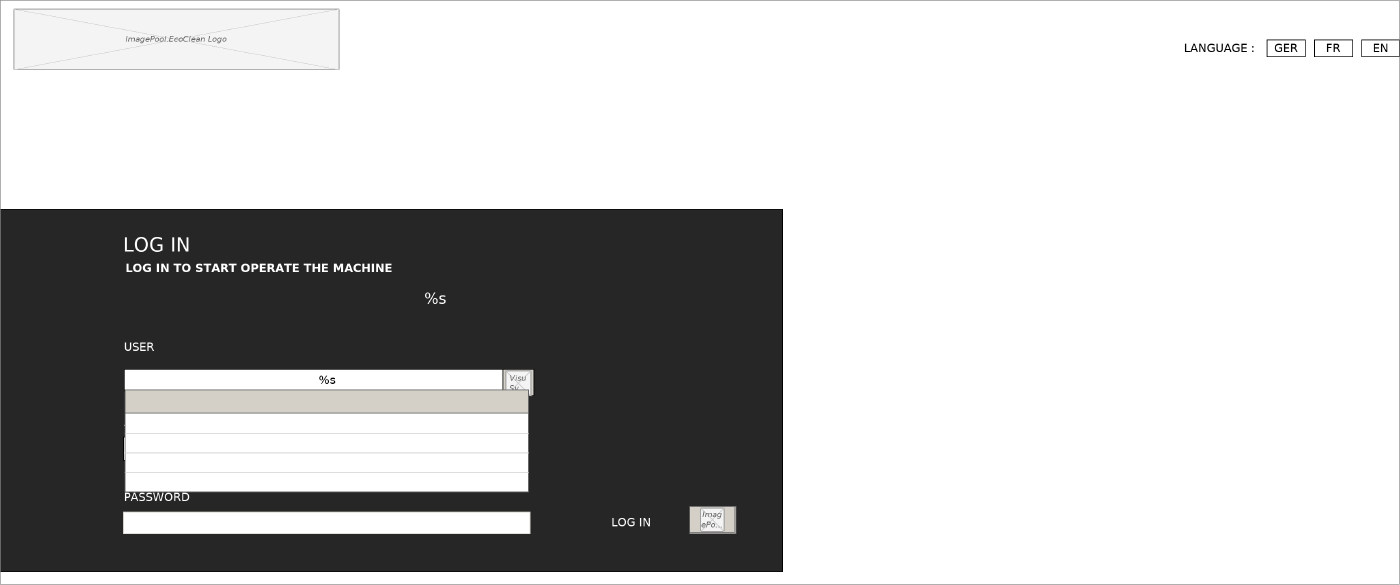
VISUALIZATION Login_Page  // 1775x742
    Label (1498,52 112x18), "LANGUAGE :"
    Rectangle (1606,50 49x22), "GER"
        OnMouseDown: ChangeLanguage ChangeLanguage=German
    Rectangle (0,252 1x490)
        p3528305787: HMI_Ctrl.ANIMATION2
    Rectangle (0,265 992x460)
    Label (153,284 221x53), "LOG IN"
    Label (156,321 609x38), "LOG IN TO START OPERATE THE MACHINE"
    Label (154,604 216x53), "PASSWORD"
    Textfield (156,649 516x28), text variable: sPasswordField
        OnMouseDown: write the text variable via Default, password
    Label (154,409 123x62), "USER"
    Label (154,509 216x53), "ACCESS LEVEL"
    Group (874,642 59x35)
        toggle bLoginPB
        Button (0,0 59x35)
        Image (14,2 30x30), image: ImagePool.Log In
    Label (733,639 135x47), "LOG IN"
    Group (157,468 516x28)
        toggle bUserNameLoginPageOn
        Rectangle (0,0 516x28), "%s", text variable: fbHmiTF1800_UserlevelManagement.dsHmiUserReg.ARsLoginName[iLoginNameId]
        Group (480,0 35x28)
            Rectangle (0,0 40x34)
            Image (4,2 32x32), image: VisuSymbols.Symbols.TriangleDown
    Textfield (168,364 768x30), "%s", text variable: sMessage
    Rectangle (156,554 513x30), "%s", text variable: fbHmiTF1800_UserlevelManagement.dsHmiUserReg.ARwsUserGroupName[iLoginNameId]
    Table (158,494 512x130), invisible if: NOT bUserNameLoginPageOn, data array: fbHmiTF1800_UserlevelManagement.dsHmiUserReg.ARsLoginName
        p3854506369: fbHmiTF1800_UserlevelManagement.dsHmiUserReg.ARsLoginName[INDEX]
        p2232123230: Login Name
        p1137915858: iLoginNameId
        Columns.Column.[0].Template: toggle bUserNameLoginPageOn
    Image (17,11 413x77), image: ImagePool.EcoClean Logo
    Rectangle (1666,50 49x22), "FR"
        OnMouseDown: ChangeLanguage ChangeLanguage=France
    Rectangle (1726,50 49x22), "EN"
        OnMouseDown: ChangeLanguage ChangeLanguage=English
END_VISUALIZATION

(* stored: Version 1.1.0.1, ProductVersion 3.1.4024.12
   Visu Login_Page: Id {add23164-a52b-4edc-849c-75c8d2c0bc4f} *)
